{attribute addProperty BoxType "EPP5101-0002-0016"}
{attribute addProperty Id "ControlAT %Q*Control_5DF70A111621Set_counter_valueAT %Q*UINT16217"}
{attribute addProperty CRC "826713010"}
{attribute addProperty SizeInBites "32"}
{attribute addProperty SizeInBytes "4"}
TYPE ENC_Control_compact_3146A3B2 :
STRUCT
	{attribute addProperty Name "Control"}
	Control AT %Q* : Control_5DF70A11;
	{attribute addProperty Name "Set_counter_value"}
	Set_counter_value AT %Q* : UINT;
END_STRUCT
END_TYPE

(* stored: Version 1.2.0.0, ProductVersion 3.1.4024.9
   DUT ENC_Control_compact_3146A3B2: Id {f0e59b2e-79cc-4bc5-a694-7ae14d38857b} *)
